PROGRAM MAIN
VAR
	bS1 : BOOL; //Schakelaar alarm aan
	bS2 : BOOL; //Bewegins detectie
	bS3 : bool; //Reset
	
	bL1 : BOOL; //Een lamp om te tonen dat het alarm aan is
	bL2 : BOOL; //Alarm
END_VAR

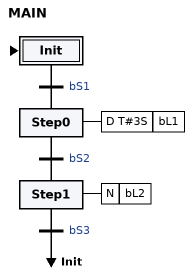
INITIAL_STEP Init:
END_STEP
TRANSITION FROM Init TO Step0
    := bS1;
END_TRANSITION
STEP Step0:
    bL1(D, T#3S);
END_STEP
TRANSITION FROM Step0 TO Step1
    := bS2;
END_TRANSITION
STEP Step1:
    bL2(N);
END_STEP
TRANSITION FROM Step1 TO Init
    := bS3;
END_TRANSITION

END_PROGRAM

(* stored: Version 1.1.0.1, ProductVersion 3.1.4024.12
   POU MAIN: Id {3d16278b-c665-443a-9423-c750f0f30854}, SpecialFunc None *)
